PROGRAM Task2
VAR
	PRG_Koffie: INT;
	bKoffieStart: BOOL;
END_VAR

// Start koffie-proces alleen als we in Deventer zijn
IF bInDeventer AND NOT bKoffieStart THEN
    bKoffieStart := TRUE;
    sStatusTekst := 'Koffie halen is gestart...';
END_IF

// Koffie ophalen (simulatie)
IF bKoffieStart THEN
    bKoffieGereed := TRUE;
    sStatusTekst := 'Koffie is gehaald!';
END_IF

END_PROGRAM

(* stored: Version 1.1.0.1, ProductVersion 3.1.4024.15
   POU Task2: Id {883ce240-6c78-41c5-9373-d8c5b7d042ae}, SpecialFunc None *)
